Staubli VAL3: empty2dNum.pgx

public program empty2dNum(num& x_nBuffer[] (dimensions=2))
  local num l_nIndex
  local num l_nIndex2
begin

  //empty a bidimensional array of num

  for l_nIndex=0 to size(x_nBuffer,1)-1
    for l_nIndex2=0 to size(x_nBuffer,2)-1
      x_nBuffer[l_nIndex,l_nIndex2]=0
    endFor
  endFor

end
